{library PUBLIC}
(* Station number type *)
TYPE StationType : INT(1..9);
END_TYPE

(* stored: Version 1.1.0.1, ProductVersion 3.1.4024.2
   EnumerationTextList StationType: Id {7e416fb9-7349-40de-9bb9-0c4415f97ae0} *)
